TYPE ST_RV_les_Stellwert :
STRUCT
	Ventil_Stellung	: REAL;
END_STRUCT
END_TYPE

(* stored: Version 1.1.0.1, ProductVersion 3.1.4024.9
   DUT ST_RV_les_Stellwert: Id {c4cd6bff-43c0-4bf7-b077-f97edd21bee8} *)
